PROGRAM MAIN
VAR
END_VAR

END_PROGRAM

(* stored: Version 1.1.0.1
   POU MAIN: Id {35c6da44-5452-4ccc-8d2a-b5b2c5d3f37b} *)
